Universal Robots PolyScope program: move_path_cover_left.urp

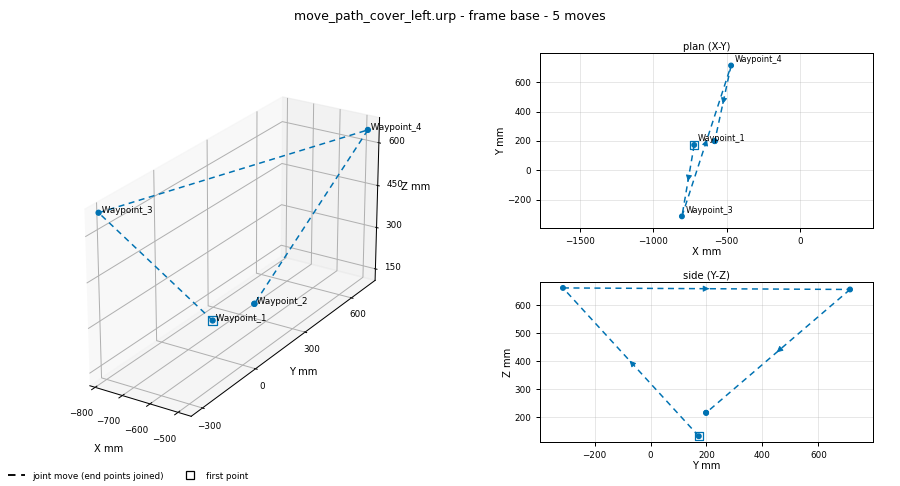
[picture p0: tool path of move_path_cover_left.urp in frame base, 5 of 17 moves have a stored position in this frame; points joined in program order, loops and branches not executed]
Program move_path_cover_left (installation=default directory=/programs createdIn=5.21.3 lastSavedIn=5.21.3 robotSerialNumber=20246801938)
Calibrated DH parameters: a=[-0.000071, -0.790281, -0.600694, 0.000061, -0.000039, 0]; d=[0.236272, 604.465945, 132.116513, -736.382239, 0.159268, 0.154005]; alpha=[1.570254, -0.000567, 0.000559, 1.571709, -1.56999, 0]; deltaTheta=[0, -0.409357, 7.293326, -0.600784, -0.000001, -0.000001]
InitVariablesNode
Robot Program (runOnlyOnce=false)
  ''
  Script: align_for_cover_left()
  Set NoAction tcp=backofhole
  ''
  p1 := pathturn[0]
  p2 := pathturn[1]
  p3 := pathturn[2]
  p4 := pathturn[3]
  p5 := pathturn[4]
  pa1 := p[p1[0],p1[1],p1[2]+0.05,p1[3],p1[4],p1[5]]
  MoveJ speed 60 deg/s, acceleration 80 deg/s^2 (useActiveTCP=true optimoveEnabled=false optiMoveSpeed=0.3 optiMoveAcceleration=0.09) feature=Base
    Waypoint Variable (Variable): variable(name=pa1)
  MoveL speed 50 mm/s, acceleration 50 mm/s^2 (useActiveTCP=true optimoveEnabled=false optiMoveSpeed=0.3 optiMoveAcceleration=0.09) feature=Base
    Waypoint Variable (Variable): variable=p1
  Wait Sleep waitTime=8
  Folder turn ext on
    URCap WireTank Serial (WireTank Serial, WireTank, LLC) dataModel(NODE_TITLE=Serial Bridge uR1, Command=[252,82,49], QUERY=false, byte_array=true, OUTPUT_ENTRY=Static, Variable(key=OUTPUT_VARIABLE, variable(name=HwResp)))
    URCap WireTank Serial (WireTank Serial, WireTank, LLC) dataModel(NODE_TITLE=Serial Bridge uR1, Command=[252,82,49], QUERY=false, byte_array=true, OUTPUT_ENTRY=Static, Variable(key=OUTPUT_VARIABLE, variable(name=HwResp)))
    Wait Sleep waitTime=1
    SuppressedNode
      Script: turn_extrusion_on()
    Set DigitalOutput pin=digital_out[0]; digitalValue=1
  MoveL speed 10 mm/s, acceleration 100 mm/s^2 (useActiveTCP=true optimoveEnabled=false optiMoveSpeed=0.3 optiMoveAcceleration=0.09) feature=Base
    Waypoint Variable (Variable): variable=p2
  MoveP speed 0.5 mm/s, acceleration 10 mm/s^2 (blendRadius=0.001 useActiveTCP=true optimoveEnabled=false optiMoveSpeed=0.3 optiMoveAcceleration=0.09) feature=Base
    CircleMove (OrientationMode=FIXED)
      Waypoint Variable (Variable): variable=p3
      Waypoint Variable (Variable): variable=p4
  MoveL speed 12 mm/s, acceleration 50 mm/s^2 (useActiveTCP=true optimoveEnabled=false optiMoveSpeed=0.3 optiMoveAcceleration=0.09) feature=Base
    Waypoint Variable (Variable): variable=p5
  URCap WireTank Serial (WireTank Serial, WireTank, LLC) dataModel(QUERY=false, NODE_TITLE=Serial Bridge uR0, Command=[252,82,48], byte_array=true, OUTPUT_ENTRY=Static, Variable(key=OUTPUT_VARIABLE, variable(name=HwResp)))
  Wait Sleep waitTime=2
  Set DigitalOutput pin=digital_out[0]; digitalValue=0
  ''
  pret1 := p[p5[0]+0.05,p5[1],p5[2],p5[3],p5[4],p5[5]]
  pret2 := p[p5[0]+0.1,p5[1],p5[2]+0.2,p5[3],p5[4],p5[5]]
  SuppressedNode
    pret2 := p[p5[0],p5[1],p5[2]-0.05,0,0,3.5]
  SuppressedNode
    p_1 := pathturn[4]
  SuppressedNode
    p_2 := pathturn[5]
  SuppressedNode
    p3 := pathturn[6]
  SuppressedNode
    p_4 := pathturn[7]
  SuppressedNode
    p_5 := pathturn[8]
  p201 := pathturn[5]
  p202 := pathturn[6]
  pret3 := p[p201[0],p201[1],p201[2]+0.05,p201[3],p201[4],p201[5]]
  pret4 := p[p202[0],p202[1],p202[2]+0.05,p202[3],p202[4],p202[5]]
  SuppressedNode
    p_preheat := p[p_3[0]+.01,p_3[1],p_3[2],p_3[3],p_3[4],p_3[5]]
  SuppressedNode
    p_pre_ret := p[p_1[0]+.03,p_1[1]+.03,p_1[2],p_1[3],p_1[4],p_1[5]]
  SuppressedNode
    p_pre_ret2 := p[p_3[0]+.1,p_3[1],p_3[2],p_3[3],p_3[4],p_3[5]]
  Set NoAction tcp=pretend_welder
  MoveL speed 50 mm/s, acceleration 50 mm/s^2 (useActiveTCP=true optimoveEnabled=false optiMoveSpeed=0.3 optiMoveAcceleration=0.09) feature=Base
    Waypoint Variable (Variable): variable=pret1
  MoveJ speed 60 deg/s, acceleration 80 deg/s^2 (useActiveTCP=true optimoveEnabled=false optiMoveSpeed=0.3 optiMoveAcceleration=0.09) feature=Base
    Waypoint Variable (Variable): variable=pret2
  MoveJ speed 60 deg/s, acceleration 80 deg/s^2 (useActiveTCP=true optimoveEnabled=false optiMoveSpeed=0.3 optiMoveAcceleration=0.09) feature=Base
    'retreat of p5'
    Waypoint Waypoint_1: TCP in base x=-720.289 y=172.595 z=132.697 mm, rx=-1.4766 ry=-0.6328 rz=0.6328 rad; joints [-143.458, -120.759, -130.403, -108.889, 80.181, 90.03] deg; TCP offset x=4.51 y=-328 z=105.73 mm, rx=1.2092 ry=-1.2092 rz=1.2092 rad
  SuppressedNode
    MoveJ speed 60 deg/s, acceleration 80 deg/s^2 (useActiveTCP=true optimoveEnabled=false optiMoveSpeed=0.3 optiMoveAcceleration=0.09) feature=Base
      Waypoint dummypoint: TCP in base x=-1096.486 y=198.657 z=80.338 mm, rx=2.9721 ry=-0.9596 rz=0.0188 rad; joints [-23.586, -40.373, 58.89, -17.461, -77.751, -1.037] deg
      Waypoint dummyret4p202: TCP in base x=-1167.172 y=17.493 z=106.65 mm, rx=2.9049 ry=-1.1452 rz=0.017 rad; joints [-16.683, -39.669, 55.352, -14.524, -63.609, -1.327] deg
  MoveJ speed 60 deg/s, acceleration 80 deg/s^2 (useActiveTCP=true optimoveEnabled=false optiMoveSpeed=0.3 optiMoveAcceleration=0.09) feature=Base
    'requires a shoulder flip. safe waypoints for that:'
    Waypoint Waypoint_3: TCP in base x=-803.735 y=-312.896 z=662.625 mm, rx=-1.3299 ry=-0.4995 rz=2.1285 rad; joints [-113.086, -77.048, -126.559, -100.277, 55.681, 86.589] deg
    Waypoint Waypoint_4: TCP in base x=-469.357 y=713.019 z=657.124 mm, rx=-2.0167 ry=1.6429 rz=0.9571 rad; joints [-73.643, -94.492, 87.56, -37.789, -83.496, -4.353] deg
  MoveJ speed 60 deg/s, acceleration 80 deg/s^2 (useActiveTCP=true optimoveEnabled=false optiMoveSpeed=0.3 optiMoveAcceleration=0.09) feature=Base
    'approach of p201'
    Waypoint Waypoint_2: TCP in base x=-580.457 y=198.657 z=216.368 mm, rx=2.9721 ry=-0.9596 rz=0.0188 rad; joints [-37.278, -75.008, 105.481, -29.448, -91.434, -0.801] deg
  MoveJ speed 60 deg/s, acceleration 80 deg/s^2 (useActiveTCP=true optimoveEnabled=false optiMoveSpeed=0.3 optiMoveAcceleration=0.09) feature=Base
    Waypoint Variable (Variable): variable=pret3
  MoveL speed 50 mm/s, acceleration 50 mm/s^2 (useActiveTCP=true optimoveEnabled=false optiMoveSpeed=0.3 optiMoveAcceleration=0.09) feature=Base
    Waypoint Variable (Variable): variable=p201
  Wait Sleep waitTime=6
  Folder turn ext on
    URCap WireTank Serial (WireTank Serial, WireTank, LLC) dataModel(NODE_TITLE=Serial Bridge uR1, Command=[252,82,49], QUERY=false, byte_array=true, OUTPUT_ENTRY=Static, Variable(key=OUTPUT_VARIABLE, variable=HwResp))
    URCap WireTank Serial (WireTank Serial, WireTank, LLC) dataModel(NODE_TITLE=Serial Bridge uR1, Command=[252,82,49], QUERY=false, byte_array=true, OUTPUT_ENTRY=Static, Variable(key=OUTPUT_VARIABLE, variable=HwResp))
    Wait Sleep waitTime=1
    SuppressedNode
      Script: turn_extrusion_on()
    Set DigitalOutput pin=digital_out[0]; digitalValue=1
  MoveL speed 12 mm/s, acceleration 100 mm/s^2 (useActiveTCP=true optimoveEnabled=false optiMoveSpeed=0.3 optiMoveAcceleration=0.09) feature=Base
    Waypoint Variable (Variable): variable=p202
  URCap WireTank Serial (WireTank Serial, WireTank, LLC) dataModel(QUERY=false, NODE_TITLE=Serial Bridge uR0, Command=[252,82,48], byte_array=true, OUTPUT_ENTRY=Static, Variable(key=OUTPUT_VARIABLE, variable=HwResp))
  Wait Sleep waitTime=2
  Set DigitalOutput pin=digital_out[0]; digitalValue=0
  MoveJ speed 60 deg/s, acceleration 80 deg/s^2 (useActiveTCP=true optimoveEnabled=false optiMoveSpeed=0.3 optiMoveAcceleration=0.09) feature=Base
    Waypoint Variable (Variable): variable=pret4
  MoveJ speed 60 deg/s, acceleration 80 deg/s^2 (useActiveTCP=true optimoveEnabled=false optiMoveSpeed=0.3 optiMoveAcceleration=0.09) feature=Base
    Waypoint Waypoint_2: TCP in base x=-580.457 y=198.657 z=216.368 mm, rx=2.9721 ry=-0.9596 rz=0.0188 rad; joints [-37.278, -75.008, 105.481, -29.448, -91.434, -0.801] deg
  SafeHome (positionOptionType=SPEED_AND_ACCELERATION speed=1.047198 acceleration=1.396263 nextMotionTime=2)
  URCap MachineLogic for Universal Robots (MachineLogic for Universal Robots, Vention Inc.) dataModel(type=addMotor, numberAdded=0, combo1=MachineMotion1, combo2=(1) Custom Actuator, combo3=Home, combo6=In series, speed_in_mm_per_min=600, acceleration_in_mm_per_s2=50.0, message=Homing, description=Moves the actuator in the negative direction until the home sensor is triggered and sets position to zero (0)., comboAddress=Address 1, comboActuator=Valve 1, teachColor=BLUE)
